Staubli VAL3: Control_Panel.pgx

program Control_Panel(string x_sTitle)
  local num l_nIndex
  local string l_sS
begin
  //画框函数
  //如果标题为空，



    setTextMode(0)

  //方框进行重画

  //画上边
   gotoxy(nPanelLTopX,nPanelLTopY)
   l_sS="┌"+left("───────────────────────────────────",nPanelWidthX)

  //写标题

     //2是两个标志符
  if x_sTitle!=""
    x_sTitle=left(x_sTitle,min(getDisplayLen(x_sTitle),nPanelWidthX)-getDisplayLen(x_sTitle)+len(x_sTitle))
    x_sTitle="┤"+x_sTitle+"├┐"
    l_sS=left(l_sS,nPanelWidthX-getDisplayLen(x_sTitle)+2)+x_sTitle
  else
    l_sS=l_sS+"┐"
  endIf
  put(l_sS)

   //画下边
   gotoxy(nPanelLTopX,nPanelLTopY+nPanelLengthY+1)
   put("└"+left("─────────────────────────────────────────",nPanelWidthX)+"┘")

   //重画两边
   for l_nIndex=1 to nPanelLengthY
    gotoxy(nPanelLTopX,nPanelLTopY+l_nIndex)
   // put("│")
   put("│")
    gotoxy(nPanelLTopX+nPanelWidthX+1,nPanelLTopY+l_nIndex)
    put("│")
  endFor












end
